FUNCTION_BLOCK IMG_CONTAINER (* Basic FB with empty ECC *)
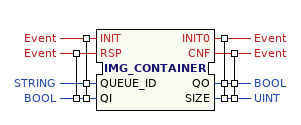
  EVENT_INPUT
    INIT WITH QUEUE_ID, QI;
    RSP WITH QI;
  END_EVENT
  EVENT_OUTPUT
    INIT0 WITH QO, SIZE;
    CNF WITH QO, SIZE;
  END_EVENT
  VAR_INPUT
    QUEUE_ID : STRING;
    QI : BOOL;
  END_VAR
  VAR_OUTPUT
    QO : BOOL;
    SIZE : UINT;
  END_VAR
END_FUNCTION_BLOCK
